TYPE ScriblyComRequest :
STRUCT
  Start : BOOL;
  Stop : BOOL;
  GoHome : BOOL;
  Halt : BOOL;
END_STRUCT
END_TYPE

(* stored: Version 1.1.0.1
   DUT ScriblyComRequest: Id {f2d5c168-a45a-4780-8a55-45d0cd021646} *)
